TYPE (* logiBUS DO Struct Dual *)
  (* Version 1.0, 2026-05-28, franz *)
  PACKAGE logiBUS::io::DQ;
  IMPORT logiBUS::io::DQ::logiBUS_DO_S;
  logiBUS_DO_S_Dual : STRUCT
    Up : logiBUS_DO_S := (Pin := 255); (* forward, up, right, clockwise *)
    Down : logiBUS_DO_S := (Pin := 255); (* backward, down, left, counter-clockwise *)
  END_STRUCT;
END_TYPE
